// TIA Portal V20 export
// export: Created 2026-08-12T15:43:40.9356965Z, ExportSetting WithDefaults, DisplayName Totally Integrated Automation Portal, DisplayVersion V20 Update 5, DisplayName TIA Portal Openness, DisplayVersion V20 Update 4, DisplayName TIA Portal Version Control Interface, DisplayVersion V20 Update 5, DisplayName SINAMICS Startdrive Advanced, DisplayVersion V20, DisplayName SINAMICS DCC, DisplayVersion V20, DisplayName SINAMICS Startdrive G130, G150, S120, S150, SINAMICS MV, G220, S200, S210, DisplayVersion V20, DisplayName SINAMICS Startdrive G110M, G120, G120C, G120D, G120P, G115D, DisplayVersion V20, DisplayName STEP 7 Professional, DisplayVersion V20 Update 5, DisplayName STEP 7 Safety, DisplayVersion V20 Update 2, DisplayName WinCC Basic/Comfort/Advanced, DisplayVersion V20 Update 5, DisplayName WinCC Unified, DisplayVersion V20 Update 5
FUNCTION "FC_FixedShapeSample" : Void   // FC8, LAD
{ S7_Optimized_Access := 'TRUE' }
VERSION : 0.1
// stored: AutoNumber true, IsIECCheckEnabled false, SetENOAutomatically false, UDAEnableTagReadback false
   VAR_TEMP
      Null : Byte;
      Req : Bool;
   END_VAR
BEGIN

REGION Network 1
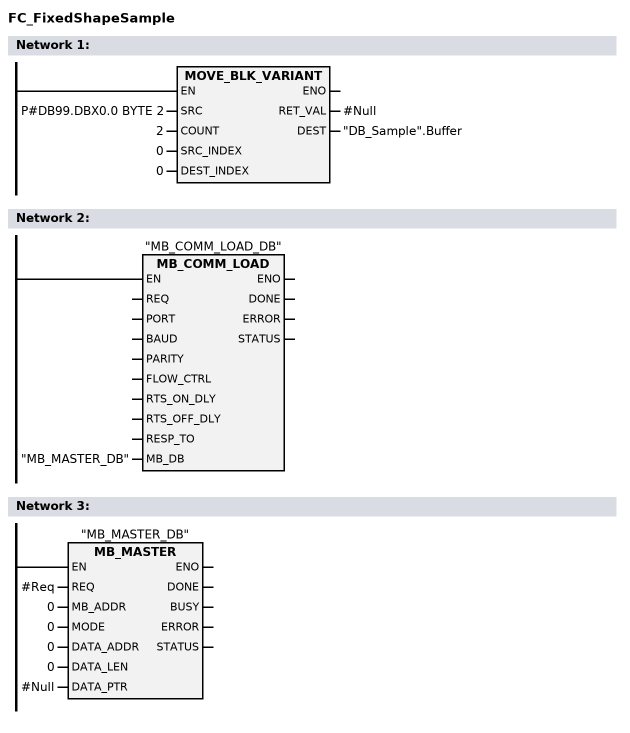
   RUNG wire#powerrail
      MOVE_BLK_VARIANT(SRC := P#DB99.DBX0.0 BYTE 2, COUNT := 2, SRC_INDEX := 0, DEST_INDEX := 0, Ret_Val => #Null, DEST => "DB_Sample".Buffer)
   END_RUNG
   // the same network as SCL:
   #Null := MOVE_BLK_VARIANT(SRC := P#DB99.DBX0.0 BYTE 2,
                           COUNT := 2,
                           SRC_INDEX := 0,
                           DEST_INDEX := 0,
                           DEST => "DB_Sample".Buffer);
END_REGION

REGION Network 2
   RUNG wire#powerrail
      "MB_COMM_LOAD_DB".MB_COMM_LOAD(REQ :=, PORT :=, BAUD :=, PARITY :=, FLOW_CTRL :=, RTS_ON_DLY :=, RTS_OFF_DLY :=, RESP_TO :=, MB_DB := "MB_MASTER_DB", DONE =>, ERROR =>, STATUS =>)
   END_RUNG
   // the same network as SCL:
   "MB_COMM_LOAD_DB"(MB_DB := "MB_MASTER_DB");   // MB_COMM_LOAD
END_REGION

REGION Network 3
   RUNG wire#powerrail
      "MB_MASTER_DB".MB_MASTER(REQ := #Req, MB_ADDR := 0, MODE := 0, DATA_ADDR := 0, DATA_LEN := 0, DATA_PTR := #Null, DONE =>, BUSY =>, ERROR =>, STATUS =>)
   END_RUNG
   // the same network as SCL:
   "MB_MASTER_DB"(REQ := #Req, MB_ADDR := 0, MODE := 0, DATA_ADDR := 0, DATA_LEN := 0, DATA_PTR := #Null);   // MB_MASTER
END_REGION
END_FUNCTION
